// TIA Portal V20 export
TYPE "LER_typeSoftcamControlNodes"
// stored: Access Published
   STRUCT
      inPos : Bool;
      isBefore : Bool;
      isAfter : Bool;
   END_STRUCT;
END_TYPE
